// TIA Portal project "string_tanimlama" (V18)

(* hardware
DEVICE "S7-1200 station_1"  S7-1200 Station
   slot 0: "Rack_0"  S7-1200 Rack  Rack  V1.0
   slot 1: "PLC_1"  CPU 1214C AC/DC/Rly  6ES7 214-1BG40-0XB0  V4.6
*)

// ===== PLC "PLC_1"  CPU 1214C AC/DC/Rly =====

VAR_GLOBAL   // PLC tag table "Default tag table"
   "Tag_1" AT %Q0.0 : Bool;
END_VAR

DATA_BLOCK "Data_block_1"   // DB1
{ S7_Optimized_Access := 'TRUE' }
VERSION : 0.1
   VAR
      İSİM : String := 'METIN_KIYAR';
      YAZILACAK_KOD : String := 'A1234DSDFHKLH';
      OKUNACAK_KOD : String;
   END_VAR
BEGIN
END_DATA_BLOCK

ORGANIZATION_BLOCK "Main"   // OB1, LAD, ProgramCycle
TITLE = "Main Program Sweep (Cycle)"
{ S7_Optimized_Access := 'TRUE' }
VERSION : 0.1
   VAR_INPUT
      Initial_Call : Bool;   // Initial call of this OB
      Remanence : Bool;   // =True, if remanent data are available
   END_VAR
BEGIN

REGION Network 1
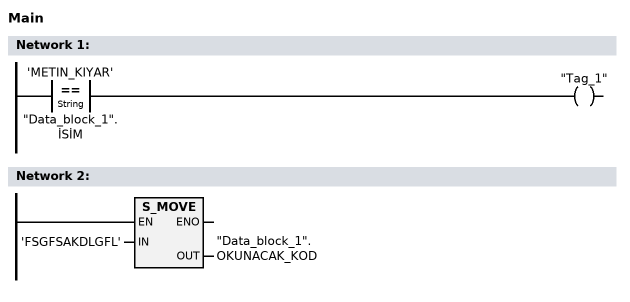
   RUNG wire#powerrail
      { S7_Templates := "SrcType := String" } EQ_Contact(in1 := 'METIN_KIYAR', in2 := "Data_block_1".İSİM)
      Coil( "Tag_1" )
   END_RUNG
   // the same network as SCL:
   "Tag_1" := 'METIN_KIYAR' = "Data_block_1".İSİM;
END_REGION

REGION Network 2
   RUNG wire#powerrail
      S_Move(in := 'FSGFSAKDLGFL', out => "Data_block_1".OKUNACAK_KOD)
   END_RUNG
   // the same network as SCL:
   "Data_block_1".OKUNACAK_KOD := 'FSGFSAKDLGFL';
END_REGION
END_ORGANIZATION_BLOCK